// LS Electric XG5000 project: 태양광완성1
// PLC LSPLC

PROGRAM NewProgram (task: 스캔 프로그램)

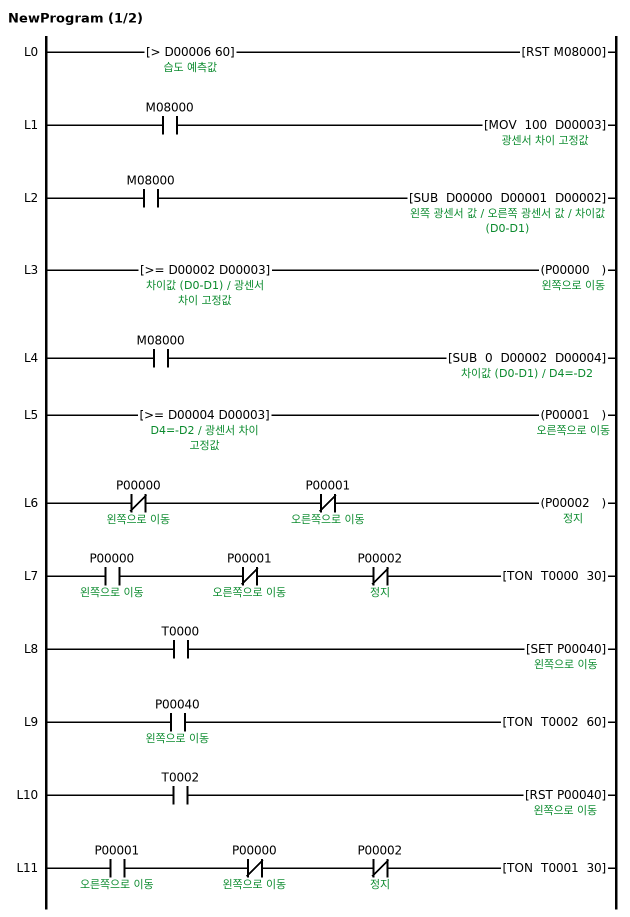
; L0
LOAD>     D00006 60	// 습도 예측값 
RST       M08000
; L1
LOAD      M08000
MOV       100 D00003	// 광센서 차이 고정값
; L2
LOAD      M08000
SUB       D00000 D00001 D00002	// 왼쪽 광센서 값 / 오른쪽 광센서 값 / 차이값 (D0-D1)
; L3
LOAD>=    D00002 D00003	// 차이값 (D0-D1) / 광센서 차이 고정값
OUT       P00000	// 왼쪽으로 이동
; L4
LOAD      M08000
SUB       0 D00002 D00004	// 차이값 (D0-D1) / D4=-D2
; L5
LOAD>=    D00004 D00003	// D4=-D2 / 광센서 차이 고정값
OUT       P00001	// 오른쪽으로 이동
; L6
LOAD NOT  P00000	// 왼쪽으로 이동
AND NOT   P00001	// 오른쪽으로 이동
OUT       P00002	// 정지
; L7
LOAD      P00000	// 왼쪽으로 이동
AND NOT   P00001	// 오른쪽으로 이동
AND NOT   P00002	// 정지
TON       T0000 30
; L8
LOAD      T0000
SET       P00040	// 왼쪽으로 이동
; L9
LOAD      P00040	// 왼쪽으로 이동
TON       T0002 60
; L10
LOAD      T0002
RST       P00040	// 왼쪽으로 이동
; L11
LOAD      P00001	// 오른쪽으로 이동
AND NOT   P00000	// 왼쪽으로 이동
AND NOT   P00002	// 정지
TON       T0001 30

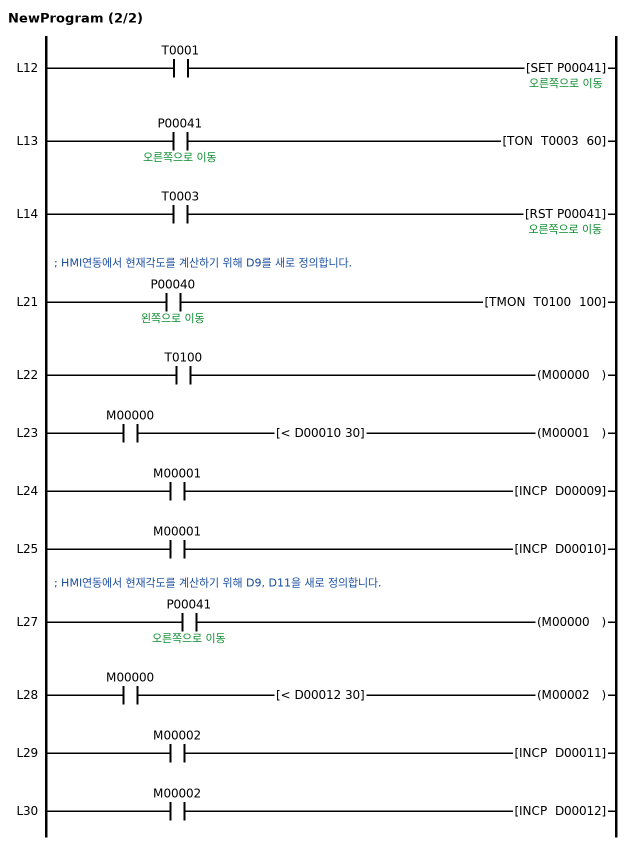
; L12
LOAD      T0001
SET       P00041	// 오른쪽으로 이동
; L13
LOAD      P00041	// 오른쪽으로 이동
TON       T0003 60
; L14
LOAD      T0003
RST       P00041	// 오른쪽으로 이동
// HMI연동에서 현재각도를 계산하기 위해 D9를 새로 정의합니다.
; L21
LOAD      P00040	// 왼쪽으로 이동
TMON      T0100 100
; L22
LOAD      T0100
OUT       M00000
; L23
LOAD      M00000
AND<      D00010 30
OUT       M00001
; L24
LOAD      M00001
INCP      D00009
; L25
LOAD      M00001
INCP      D00010
// HMI연동에서 현재각도를 계산하기 위해 D9, D11을 새로 정의합니다.
; L27
LOAD      P00041	// 오른쪽으로 이동
OUT       M00000
; L28
LOAD      M00000
AND<      D00012 30
OUT       M00002
; L29
LOAD      M00002
INCP      D00011
; L30
LOAD      M00002
INCP      D00012

VARIABLES AND COMMENTS (devices not used above)
P00042	BIT	정지